PROGRAM slave
VAR
	axis: AXIS_REF;
	
	mcPower: MC_Power;
	shouldPowerOn: BOOL;
	isMotorReady: BOOL;
	
	mcSetPosition: MC_SetPosition;
	shouldSetZero: BOOL;
END_VAR

METHOD checkPower : BOOL
VAR_INPUT
END_VAR
mcPower(
	Axis:= axis, 
	Enable:= shouldPowerOn, 
	Enable_Positive:= TRUE, 
	Enable_Negative:= TRUE,
	Status=> isMotorReady
);
END_METHOD

ACTION checkSetPoint:
mcSetPosition(
	Axis:= axis, 
	Execute:= shouldSetZero,
	Position := 0);
END_ACTION

ACTION dummyAction:

END_ACTION

END_PROGRAM

(* stored: Version 1.1.0.1, ProductVersion 3.1.4024.4
   POU slave: Id {dbf4b02e-4599-4618-990b-b48c5a0ba3e6}, SpecialFunc None
   Method checkPower: Id {2379a7cf-6f88-4d52-a90b-2cfc7a819242}
   Action checkSetPoint: Id {6c975783-f282-40f4-889b-29d37e819d33}
   Action dummyAction: Id {585f1df4-8173-4897-a8cd-909d3cbfbcc2} *)
